(* CODESYS project tcl_SimpleUnitTestLibrary.library
   Company: Red Rock Controls Limited
   Description: Local variables in T_UnitTestBase hidden
   Version: 1.1.10.2
   Placeholder: tcl_SimpleUnitTestLibrary
   Author: Roger Christopher
   Title: tcl_SimpleUnitTestLibrary

Project tree, tasks and I/O mapping:
  libraries: Tc2_EtherCAT, * (Beckhoff Automation GmbH); Tc2_Standard, * (Beckhoff Automation GmbH); Tc2_System, * (Beckhoff Automation GmbH); Tc2_Utilities, * (Beckhoff Automation GmbH); Tc3_Module, * (Beckhoff Automation GmbH); tcl_StringUtils, * (Red Rock Controls Limited)
  GVLs/
    global variables Parameters
  Unit Test Framework/
    Assertions/
      interface I_AssertionMessageList: AddMessage, Clear
      function block T_Assertion [ST]: Assert, AssertEquals_BLOB, AssertEquals_BOOL, AssertEquals_BYTE, AssertEquals_DINT, AssertEquals_DWORD, AssertEquals_INT, AssertEquals_INTERFACE, AssertEquals_LINT, AssertEquals_LREAL, AssertEquals_PVOID, AssertEquals_REAL, AssertEquals_STRING, AssertEquals_UDINT, AssertEquals_UINT, AssertEquals_ULINT, AssertEquals_WORD, AssertNotEquals_INTERFACE, FB_init, AssertionFailed, AssertionMessage
    Message list/
      function block T_AssertionMessageList [ST]: AddMessage, Clear, FB_init
    Test Runner/
      Test Runner/
        function block T_TestRunner [ST]: AddTest, AddTestSuite, BeginTesting, ClearTests, DisableAll, EnableAll, GetEnabledTestCount, GetResultsSummary, Initialisation, ResetTests, ToggleTestEnable, Busy, ReloadTests, TestFinished
    TestSuite/
      interface I_TestSuite: AddTest, GetTest, Name, TestCount
      function block T_TestSuite [ST]: AddTest, FB_init, GetTest, Name, TestCount
    Unit Test/
      interface I_AssertionListener: OnAssertionFailed, TestName
      interface I_UnitTest: Execute, Initialise, CompletedTestsCount, FailedTestsCount, ImageRef, SuiteName, TestCompleted, TestEnabled, TestHasFailed, TestHasFinished, TestName, TestState
      function block T_UnitTestBase [ST]: Execute, FB_init, Initialise, OnAssertionFailed, setTestName, TestFinished, CompletedTestsCount, FailedTestsCount, ImageRef, SuiteName, TestCompleted, TestEnabled, TestHasFailed, TestHasFinished, TestName, TestState
    Version/
      global variables Global_Version
    data type ST_TestResult
  VISUs/
    visualisation Visualization
  GlobalImagePool
  00000000-0000-0000-0000-000000000000|Images\Failed.png
  00000000-0000-0000-0000-000000000000|Images\Passed.png
  00000000-0000-0000-0000-000000000000|Images\BlueRight.png
  text list GlobalTextList
*)

// Unit Test Framework/ST_TestResult
TYPE
    ST_TestResult :
    STRUCT
        SuiteName : T_MaxString;
        TestName  : T_MaxString;
        TestState : T_MaxString;
        ImageRef  : STRING;
    END_STRUCT
END_TYPE

// GVLs/Parameters
VAR_GLOBAL CONSTANT
    MAX_TESTS              : DINT := 200;
    MAX_ASSERTION_MESSAGES : DINT := 200;
END_VAR

// Unit Test Framework/Version/Global_Version
{attribute 'TcGenerated'}
{attribute 'no-analysis'}
{attribute 'linkalways'}
// This function has been automatically generated from the project information.
VAR_GLOBAL CONSTANT
	{attribute 'const_non_replaced'}
	stLibVersion_tcl_SimpleUnitTestLibrary : ST_LibVersion := (iMajor := 1, iMinor := 1, iBuild := 10, iRevision := 2, nFlags := 0, sVersion := '1.1.10.2');
END_VAR

// Unit Test Framework/Assertions/I_AssertionMessageList
INTERFACE I_AssertionMessageList

METHOD AddMessage : BOOL
VAR_INPUT
    Message : T_MaxString;
END_VAR
END_METHOD

METHOD Clear
VAR_INPUT
END_VAR
END_METHOD

END_INTERFACE

// Unit Test Framework/Assertions/T_Assertion
FUNCTION_BLOCK T_Assertion
VAR_INPUT
END_VAR
VAR_OUTPUT
END_VAR
VAR
    _AssertionFailed : BOOL;
    _AssertionMessage : T_MaxString;
    _ExpectedAsString : T_MaxString;
    _ActualAsString   : T_MaxString;
    _AssertionListener : I_AssertionListener;
END_VAR

METHOD Assert
VAR_INPUT
    AssertionMessage : T_MaxString;
    Expected         : T_MaxString;
    Actual           : T_MaxString;
END_VAR
_AssertionFailed := TRUE;
_AssertionMessage := F_FormatStringEx2('Assertion failed in %s - %s',_AssertionListener.TestName, AssertionMessage);
    _ExpectedAsString := F_FormatStringEx1('  Expected = %s', Expected);
    _ActualAsString   := F_FormatStringEx1('  Actual   = %s', Actual);
_AssertionListener.OnAssertionFailed(_AssertionMessage,_ExpectedAsString,_ActualAsString);
END_METHOD

METHOD AssertEquals_BLOB
VAR_INPUT
    Expected : ANY;
    Actual   : ANY;
    VariableName : T_MaxString;
END_VAR
IF Expected.diSize <> Actual.diSize THEN
    _AssertionFailed := TRUE;
    _AssertionMessage := F_FormatStringEx2('AssertEquals_BLOB failed in %s: Value "%s"', _AssertionListener.TestName, 'Blob.Size');
    _ExpectedAsString := F_FormatString1('  Expected = %d', F_DINT(Expected.diSize));
    _ActualAsString   := F_FormatString1('  Actual   = %d', F_DINT(Actual.diSize));
    _AssertionListener.OnAssertionFailed(_AssertionMessage,_ExpectedAsString,_ActualAsString);
    
ELSIF Expected.TypeClass <> Actual.TypeClass THEN
    _AssertionFailed := TRUE;
    _AssertionMessage := F_FormatStringEx2('AssertEquals_BLOB failed in %s: Value "%s"', _AssertionListener.TestName, 'Blob.TypeClass');
    _ExpectedAsString := F_FormatStringEx1('  Expected = %s', F_TypeClassToString(Expected.TypeClass));
    _ActualAsString   := F_FormatStringEx1('  Actual   = %s', F_TypeClassToString(Actual.TypeClass));
    _AssertionListener.OnAssertionFailed(_AssertionMessage,_ExpectedAsString,_ActualAsString);
    
ELSIF 
    MEMCMP(
        pBuf1 := Expected.pValue, 
        pBuf2 := Actual.pValue, 
        n     := DINT_TO_UDINT(Actual.diSize)) <> 0
THEN
    _AssertionFailed := TRUE;
    _AssertionMessage := F_FormatStringEx1('AssertEquals_BLOB failed in %s: Contents differ', _AssertionListener.TestName);
    _ExpectedAsString := '';
    _ActualAsString   := '';
    _AssertionListener.OnAssertionFailed(_AssertionMessage,_ExpectedAsString,_ActualAsString);
ELSE
    _AssertionFailed  := FALSE;
    _AssertionMessage := '';
END_IF
END_METHOD

METHOD AssertEquals_BOOL 
VAR_INPUT
    Expected : BOOL;
    Actual   : BOOL;
    VariableName : T_MaxString;
END_VAR
IF Expected <> Actual THEN
    _AssertionFailed  := TRUE;
    _AssertionMessage := F_FormatStringEx2('AssertEquals_BOOL failed in %s: Value "%s"', _AssertionListener.TestName, VariableName);
    _ExpectedAsString := F_FormatStringEx1('  Expected = %s', BOOL_TO_STRING(Expected));
    _ActualAsString   := F_FormatStringEx1('  Actual   = %s', BOOL_TO_STRING(Actual));
    _AssertionListener.OnAssertionFailed(_AssertionMessage,_ExpectedAsString,_ActualAsString);
ELSE
    _AssertionFailed   := FALSE;
    _AssertionMessage  := '';
END_IF
END_METHOD

METHOD AssertEquals_BYTE
VAR_INPUT
    Expected : BYTE;
    Actual   : BYTE;
    VariableName : T_MaxString;
END_VAR
IF Expected <> Actual THEN
    _AssertionFailed := TRUE;
    _AssertionMessage := F_FormatStringEx2('AssertEquals_BYTE failed in %s: Value "%s"', _AssertionListener.TestName, VariableName);
    _ExpectedAsString := F_FormatString1('  Expected = %d', F_BYTE(Expected));
    _ActualAsString   := F_FormatString1('  Actual   = %d', F_BYTE(Actual));
    _AssertionListener.OnAssertionFailed(_AssertionMessage,_ExpectedAsString,_ActualAsString);
ELSE
    _AssertionFailed  := FALSE;
    _AssertionMessage := '';
END_IF
END_METHOD

METHOD AssertEquals_DINT 
VAR_INPUT
    Expected : DINT;
    Actual   : DINT;
    VariableName : T_MaxString;
END_VAR
IF Expected <> Actual THEN
    _AssertionFailed  := TRUE;
    _AssertionMessage := F_FormatStringEx2('AssertEquals_DINT failed in %s: Value "%s"', _AssertionListener.TestName, VariableName);
    _ExpectedAsString := F_FormatString1('  Expected = %d', F_DINT(Expected));
    _ActualAsString   := F_FormatString1('  Actual   = %d', F_DINT(Actual));
    _AssertionListener.OnAssertionFailed(_AssertionMessage,_ExpectedAsString,_ActualAsString);
ELSE
    _AssertionFailed  := FALSE;
    _AssertionMessage := '';
END_IF
END_METHOD

METHOD AssertEquals_DWORD
VAR_INPUT
    Expected : DWORD;
    Actual   : DWORD;
    VariableName : T_MaxString;
END_VAR
IF Expected <> Actual THEN
    _AssertionFailed := TRUE;
    _AssertionMessage := F_FormatStringEx2('AssertEquals_DWORD failed in %s: Value "%s"', _AssertionListener.TestName, VariableName);
    _ExpectedAsString := F_FormatString1('  Expected = %d', F_DWORD(Expected));
    _ActualAsString   := F_FormatString1('  Actual   = %d', F_DWORD(Actual));
    _AssertionListener.OnAssertionFailed(_AssertionMessage,_ExpectedAsString,_ActualAsString);
ELSE
    _AssertionFailed  := FALSE;
    _AssertionMessage := '';
END_IF
END_METHOD

METHOD AssertEquals_INT
VAR_INPUT
    Expected : INT;
    Actual   : INT;
    VariableName : T_MaxString;
END_VAR
IF Expected <> Actual THEN
    _AssertionFailed := TRUE;
    _AssertionMessage := F_FormatStringEx2('AssertEquals_INT failed in %s: Value "%s"', _AssertionListener.TestName, VariableName);
    _ExpectedAsString := F_FormatString1('  Expected = %d', F_INT(Expected));
    _ActualAsString   := F_FormatString1('  Actual   = %d', F_INT(Actual));
    _AssertionListener.OnAssertionFailed(_AssertionMessage,_ExpectedAsString,_ActualAsString);
ELSE
    _AssertionFailed  := FALSE;
    _AssertionMessage := '';
END_IF
END_METHOD

METHOD AssertEquals_INTERFACE 
VAR_INPUT
    Expected : __SYSTEM.IQueryInterface;
    Actual   : __SYSTEM.IQueryInterface;
    VariableName : T_MaxString;
END_VAR
IF Expected <> Actual THEN
    _AssertionFailed  := TRUE;
    _AssertionMessage := F_FormatStringEx2('AssertEquals_INTERFACE failed in %s: Value "%s"', _AssertionListener.TestName, VariableName);
    _ExpectedAsString := '  Interfaces Differ';
    _ActualAsString   := '';
    _AssertionListener.OnAssertionFailed(_AssertionMessage,_ExpectedAsString,_ActualAsString);
ELSE
    _AssertionFailed  := FALSE;
    _AssertionMessage := '';
END_IF
END_METHOD

METHOD AssertEquals_LINT 
VAR_INPUT
    Expected : LINT;
    Actual   : LINT;
    VariableName : T_MaxString;
END_VAR
IF Expected <> Actual THEN
    _AssertionFailed  := TRUE;
    _AssertionMessage := F_FormatStringEx2('AssertEquals_LINT failed in %s: Value "%s"', _AssertionListener.TestName, VariableName);
    _ExpectedAsString := F_FormatString1('  Expected = %d', F_LINT(Expected));
    _ActualAsString   := F_FormatString1('  Actual   = %d', F_LINT(Actual));
    _AssertionListener.OnAssertionFailed(_AssertionMessage,_ExpectedAsString,_ActualAsString);
ELSE
    _AssertionFailed  := FALSE;
    _AssertionMessage := '';
END_IF
END_METHOD

METHOD AssertEquals_LREAL 
VAR_INPUT
    Expected : LREAL;
    Actual   : LREAL;
    Delta    : LREAL;
    VariableName : T_MaxString;
END_VAR
IF ABS(Expected - Actual) > Delta THEN
    _AssertionFailed  := TRUE;
    _AssertionMessage := F_FormatStringEx2('AssertEquals_LREAL failed in %s: Value "%s"', _AssertionListener.TestName, VariableName);
    _ExpectedAsString := F_FormatString1('  Expected = %f', F_LREAL(Expected));
    _ActualAsString   := F_FormatString1('  Actual   = %f', F_LREAL(Actual));
    _AssertionListener.OnAssertionFailed(_AssertionMessage,_ExpectedAsString,_ActualAsString);
ELSE
    _AssertionFailed  := FALSE;
    _AssertionMessage := '';
END_IF
END_METHOD

METHOD AssertEquals_PVOID 
VAR_INPUT
    Expected : PVOID;
    Actual   : PVOID;
    VariableName : T_MaxString;
END_VAR
IF Expected <> Actual THEN
    _AssertionFailed  := TRUE;
    _AssertionMessage := F_FormatStringEx2('AssertEquals_PVOID failed in %s: Value "%s"', _AssertionListener.TestName, VariableName);
    _ExpectedAsString := F_FormatString1('  Expected = %d', F_PVOID(Expected));
    _ActualAsString   := F_FormatString1('  Actual   = %d', F_PVOID(Actual));
    _AssertionListener.OnAssertionFailed(_AssertionMessage,_ExpectedAsString,_ActualAsString);
ELSE
    _AssertionFailed  := FALSE;
    _AssertionMessage := '';
END_IF
END_METHOD

METHOD AssertEquals_REAL 
VAR_INPUT
    Expected : REAL;
    Actual   : REAL;
    Delta    : REAL;
    VariableName : T_MaxString;
END_VAR
IF ABS(Expected - Actual) > Delta THEN
    _AssertionFailed  := TRUE;
    _AssertionMessage := F_FormatStringEx2('AssertEquals_REAL failed in %s: Value "%s"', _AssertionListener.TestName, VariableName);
    _ExpectedAsString := F_FormatString1('  Expected = %f', F_REAL(Expected));
    _ActualAsString   := F_FormatString1('  Actual   = %f', F_REAL(Actual));
    _AssertionListener.OnAssertionFailed(_AssertionMessage,_ExpectedAsString,_ActualAsString);
ELSE
    _AssertionFailed  := FALSE;
    _AssertionMessage := '';
END_IF
END_METHOD

METHOD AssertEquals_STRING
VAR_INPUT
    Expected : T_MaxString;
    Actual   : T_MaxString;
    VariableName : T_MaxString;
END_VAR
IF Expected <> Actual THEN
    _AssertionFailed := TRUE;
    _AssertionMessage := F_FormatStringEx2('AssertEquals_STRING failed in %s: Value "%s"', _AssertionListener.TestName, VariableName);
    _ExpectedAsString := F_FormatStringEx1('  Expected = %s', Expected);
    _ActualAsString   := F_FormatStringEx1('  Actual   = %s', Actual);
    _AssertionListener.OnAssertionFailed(_AssertionMessage,_ExpectedAsString,_ActualAsString);
ELSE
    _AssertionFailed   := FALSE;
    _AssertionMessage  := '';
    _ExpectedAsString  := '';
    _ActualAsString    := '';
END_IF
END_METHOD

METHOD AssertEquals_UDINT
VAR_INPUT
    Expected : UDINT;
    Actual   : UDINT;
    VariableName : T_MaxString;
END_VAR
IF Expected <> Actual THEN
    _AssertionFailed := TRUE;
    _AssertionMessage := F_FormatStringEx2('AssertEquals_UDINT failed in %s: Value "%s"', _AssertionListener.TestName, VariableName);
    _ExpectedAsString := F_FormatString1('  Expected = %d', F_UDINT(Expected));
    _ActualAsString   := F_FormatString1('  Actual   = %d', F_UDINT(Actual));
    _AssertionListener.OnAssertionFailed(_AssertionMessage,_ExpectedAsString,_ActualAsString);
ELSE
    _AssertionFailed  := FALSE;
    _AssertionMessage := '';
END_IF
END_METHOD

METHOD AssertEquals_UINT
VAR_INPUT
    Expected : UINT;
    Actual   : UINT;
    VariableName : T_MaxString;
END_VAR
IF Expected <> Actual THEN
    _AssertionFailed := TRUE;
    _AssertionMessage := F_FormatStringEx2('AssertEquals_UINT failed in %s: Value "%s"', _AssertionListener.TestName, VariableName);
    _ExpectedAsString := F_FormatString1('  Expected = %d', F_UINT(Expected));
    _ActualAsString   := F_FormatString1('  Actual   = %d', F_UINT(Actual));
    _AssertionListener.OnAssertionFailed(_AssertionMessage,_ExpectedAsString,_ActualAsString);
ELSE
    _AssertionFailed  := FALSE;
    _AssertionMessage := '';
END_IF
END_METHOD

METHOD AssertEquals_ULINT 
VAR_INPUT
    Expected : ULINT;
    Actual   : ULINT;
    VariableName : T_MaxString;
END_VAR
IF Expected <> Actual THEN
    _AssertionFailed  := TRUE;
    _AssertionMessage := F_FormatStringEx2('AssertEquals_ULINT failed in %s: Value "%s"', _AssertionListener.TestName, VariableName);
    _ExpectedAsString := F_FormatString1('  Expected = %d', F_ULINT(Expected));
    _ActualAsString   := F_FormatString1('  Actual   = %d', F_ULINT(Actual));
    _AssertionListener.OnAssertionFailed(_AssertionMessage,_ExpectedAsString,_ActualAsString);
ELSE
    _AssertionFailed  := FALSE;
    _AssertionMessage := '';
END_IF
END_METHOD

METHOD AssertEquals_WORD
VAR_INPUT
    Expected : WORD;
    Actual   : WORD;
    VariableName : T_MaxString;
END_VAR
IF Expected <> Actual THEN
    _AssertionFailed := TRUE;
    _AssertionMessage := F_FormatStringEx2('AssertEquals_WORD failed in %s: Value "%s"', _AssertionListener.TestName, VariableName);
    _ExpectedAsString := F_FormatString1('  Expected = %d', F_WORD(Expected));
    _ActualAsString   := F_FormatString1('  Actual   = %d', F_WORD(Actual));
    _AssertionListener.OnAssertionFailed(_AssertionMessage,_ExpectedAsString,_ActualAsString);
ELSE
    _AssertionFailed  := FALSE;
    _AssertionMessage := '';
END_IF
END_METHOD

METHOD AssertNotEquals_INTERFACE 
VAR_INPUT
    Expected : __SYSTEM.IQueryInterface;
    Actual   : __SYSTEM.IQueryInterface;
    VariableName : T_MaxString;
END_VAR
IF Expected = Actual THEN
    _AssertionFailed  := TRUE;
    _AssertionMessage := F_FormatStringEx2('AssertNotEquals_INTERFACE failed in %s: Value "%s"', _AssertionListener.TestName, VariableName);
    _ExpectedAsString := '  Interfaces are the same';
    _ActualAsString   := '';
    _AssertionListener.OnAssertionFailed(_AssertionMessage,_ExpectedAsString,_ActualAsString);
ELSE
    _AssertionFailed  := FALSE;
    _AssertionMessage := '';
END_IF
END_METHOD

METHOD FB_init : BOOL
VAR_INPUT
	bInitRetains : BOOL; // if TRUE, the retain variables are initialized (warm start / cold start)
	bInCopyCode : BOOL;  // if TRUE, the instance afterwards gets moved into the copy code (online change)
    AssertionListener : I_AssertionListener;
END_VAR
_AssertionListener := AssertionListener;
END_METHOD

PROPERTY AssertionFailed : BOOL
GET
AssertionFailed := _AssertionFailed;
END_GET
END_PROPERTY

PROPERTY AssertionMessage : T_MaxString
GET
AssertionMessage := _AssertionMessage;
END_GET
END_PROPERTY

END_FUNCTION_BLOCK

// Unit Test Framework/Unit Test/I_AssertionListener
INTERFACE I_AssertionListener

METHOD OnAssertionFailed
VAR_INPUT
    AssertionMessage : T_MaxString;
    ExpectedAsString : T_MaxString;
    ActualAsString   : T_MaxString;
END_VAR
END_METHOD

{attribute 'monitoring' := 'call'}
PROPERTY TestName : T_MaxString
GET
END_GET
END_PROPERTY

END_INTERFACE

// Unit Test Framework/Message list/T_AssertionMessageList
FUNCTION_BLOCK T_AssertionMessageList IMPLEMENTS I_AssertionMessageList
VAR
    Messages : REFERENCE TO ARRAY[0..MAX_ASSERTION_MESSAGES] OF T_MaxString;
    Count : INT;
END_VAR

METHOD AddMessage : BOOL
VAR_INPUT
    Message : T_MaxString;
END_VAR
IF Count <= MAX_ASSERTION_MESSAGES THEN
    Messages[Count] := Message;
    Count := Count + 1;
    AddMessage := TRUE;
END_IF
END_METHOD

METHOD Clear
VAR_INPUT
END_VAR
MEMSET(
    destAddr := ADR(Messages), 
    fillByte := 0, 
    n        := SIZEOF(Messages));
Count := 0;
END_METHOD

METHOD FB_init : BOOL
VAR_INPUT
    bInitRetains : BOOL; // if TRUE, the retain variables are initialized (warm start / cold start)
    bInCopyCode  : BOOL; // if TRUE, the instance afterwards gets moved into the copy code (online change)
    Messages     : REFERENCE TO ARRAY[0..MAX_ASSERTION_MESSAGES] OF T_MaxString;
END_VAR
THIS^.Messages REF= Messages;
END_METHOD

END_FUNCTION_BLOCK

// Unit Test Framework/Test Runner/Test Runner/T_TestRunner
FUNCTION_BLOCK T_TestRunner
VAR
    _ReloadTests         : BOOL := TRUE; // Also exposed as a property so it can be read and reset by client
    RunTestsSequentially : BOOL := TRUE;
    Run                  : BOOL;
    Reset                : BOOL;
    EnableAllTests       : BOOL;
    DisableAllTests      : BOOL;
    RowIsSelected        : BOOL;
    SelectedRow          : INT := -1;
    Abort                : BOOL;

    State : (
        Init,
        StartTests,
        RunTests_Concurrently,
        RunTests_Sequentially,
        CheckResults
    );

    i                        : DINT;
    CompletedTestsCount      : DINT;
    FailedTestsCount         : DINT;
    CurrentTestIndex         : DINT;
    TestsCompletedPercentage : LREAL;
    TestCount                : DINT;
    EnabledTestCount         : DINT;
    ResultsSummary           : T_MaxString;

    Results  : ARRAY[0..MAX_TESTS] OF ST_TestResult;
    Tests    : ARRAY[0..MAX_TESTS] OF I_UnitTest;
    Messages : ARRAY[0..MAX_ASSERTION_MESSAGES] OF T_MaxString; // must be located here so vis can access them

    AssertionMessages : T_AssertionMessageList(Messages := Messages);

END_VAR

IF RowIsSelected THEN
    ToggleTestEnable(Index := SelectedRow);
    RowIsSelected := FALSE;
	SelectedRow := -1;
END_IF

IF EnableAllTests THEN
    EnableAllTests := FALSE;
    EnableAll();
END_IF

IF DisableAllTests THEN
    DisableAllTests := FALSE;
    DisableAll();
END_IF

IF Abort THEN
	Abort := FALSE;
	State := 0;
	Initialisation();
END_IF

CASE State OF
    Init:
        IF Reset THEN
            Reset := FALSE;
            Initialisation();
        END_IF

        IF Run THEN
            Run              := FALSE;
            EnabledTestCount := GetEnabledTestCount();

            IF EnabledTestCount = 0 THEN
                State := CheckResults;
            ELSE
                State := StartTests;
            END_IF
        END_IF

    StartTests:
        IF RunTestsSequentially THEN
            State := RunTests_Sequentially;
        ELSE
            State := RunTests_Concurrently;
        END_IF

    RunTests_Concurrently:
        FOR i := 0 TO TestCount - 1 DO
            Tests[i].Execute();
			Results[i].TestState := Tests[i].TestState;
			Results[i].ImageRef  := Tests[i].ImageRef;
        END_FOR

        IF EnabledTestCount > 0 THEN
            TestsCompletedPercentage := CompletedTestsCount * 100 / EnabledTestCount;
        END_IF

        ResultsSummary := GetResultsSummary();

        IF CompletedTestsCount >= EnabledTestCount THEN
            State := CheckResults;
        END_IF

    RunTests_Sequentially:
        IF Tests[CurrentTestIndex] <> 0 THEN
            Tests[CurrentTestIndex].Execute();
			Results[CurrentTestIndex].TestState := Tests[CurrentTestIndex].TestState;
			Results[CurrentTestIndex].ImageRef  := Tests[CurrentTestIndex].ImageRef;

            IF NOT Tests[CurrentTestIndex].TestEnabled OR Tests[CurrentTestIndex].TestHasFinished THEN
                CurrentTestIndex := CurrentTestIndex + 1;
            END_IF
        END_IF

        IF EnabledTestCount > 0 THEN
            TestsCompletedPercentage := CompletedTestsCount * 100 / EnabledTestCount;
        END_IF

        ResultsSummary := GetResultsSummary();

        IF CurrentTestIndex >= TestCount THEN
            State := CheckResults;
        END_IF

    CheckResults:
        ResultsSummary := GetResultsSummary();
        State          := Init;

END_CASE

METHOD AddTest : BOOL
VAR_INPUT
    UnitTest : I_UnitTest;
END_VAR
IF TestCount < MAX_TESTS THEN
    UnitTest.TestEnabled := TRUE;
    Tests[TestCount]    := UnitTest;
	    Results[TestCount].SuiteName := UnitTest.SuiteName;
	    Results[TestCount].TestName  := UnitTest.TestName;
	    Results[TestCount].TestState := UnitTest.TestState;
	    Results[TestCount].ImageRef  := UnitTest.ImageRef;
	
    TestCount           := TestCount + 1;
    AddTest              := TRUE;
ELSE
    AssertionMessages.AddMessage('Maximum unit tests exceeded!');
END_IF
END_METHOD

METHOD AddTestSuite : BOOL
VAR_INPUT
    TestSuite : I_TestSuite;
END_VAR
VAR
    i : INT;
    UnitTestToAdd : I_UnitTest;
END_VAR
IF TestSuite.TestCount > 0 THEN
    FOR i := 0 TO TestSuite.TestCount - 1 DO
        UnitTestToAdd := TestSuite.GetTest(i);
        AddTest(UnitTestToAdd);
    END_FOR
END_IF
END_METHOD

METHOD PUBLIC BeginTesting : BOOL
IF state <> init THEN
  RETURN;
END_IF

Run := TRUE;
BeginTesting := TRUE;
END_METHOD

METHOD ClearTests
VAR_INPUT
END_VAR
FOR i := 0 TO MAX_TESTS DO
    Tests[i] := 0;
END_FOR
MEMSET(
	destAddr:= ADR(Results), 
	fillByte:= 0, 
	n:= SIZEOF(Results));
TestCount := 0;
END_METHOD

METHOD DisableAll
VAR_INPUT
END_VAR
IF State = Init THEN
    FOR i := 0 TO MAX_TESTS - 1 DO
        IF Tests[i] <> 0 THEN
            Tests[i].TestEnabled := FALSE;
			Results[i].TestState := 'Disabled';
        END_IF
    END_FOR
END_IF
END_METHOD

METHOD EnableAll
VAR_INPUT
END_VAR
IF State = Init THEN
    FOR i := 0 TO MAX_TESTS - 1 DO
        IF Tests[i] <> 0 THEN
            Tests[i].TestEnabled := TRUE;
			Results[i].TestState := 'Enabled';
        END_IF
    END_FOR
END_IF
END_METHOD

METHOD GetEnabledTestCount : DINT
VAR
    i : DINT;
END_VAR
FOR i := 0 TO MAX_TESTS - 1 DO
    IF Tests[i] <> 0 THEN
        IF Tests[i].TestEnabled THEN
            GetEnabledTestCount := GetEnabledTestCount + 1;
        END_IF
    END_IF
END_FOR
END_METHOD

METHOD GetResultsSummary : T_MaxString
VAR_INPUT
END_VAR
GetResultsSummary := F_FormatString3('%d Tests of %d completed, %d Tests Failed',
                            F_DINT(CompletedTestsCount),
                            F_DINT(EnabledTestCount),
                            F_DINT(FailedTestsCount));
END_METHOD

METHOD Initialisation
VAR_INPUT
END_VAR
VAR
    i : DINT;
END_VAR
FOR i := 0 TO MAX_TESTS DO
    IF Tests[i] <> 0 THEN
        Tests[i].Initialise(AssertionMessages,
                            CompletedTestsCount := CompletedTestsCount,
                            FailedTestsCount    := FailedTestsCount);
							
	    Results[i].SuiteName := Tests[i].SuiteName;
	    Results[i].TestName  := Tests[i].TestName;
	    Results[i].TestState := Tests[i].TestState;
	    Results[i].ImageRef  := Tests[i].ImageRef;
    END_IF
END_FOR

ResultsSummary           := '';
FailedTestsCount         := 0;
CompletedTestsCount      := 0;
TestsCompletedPercentage := 0;
CurrentTestIndex         := 0;
AssertionMessages.Clear();
END_METHOD

METHOD PUBLIC ResetTests : BOOL
VAR_INPUT
END_VAR
IF state <> Init THEN
  RETURN;
END_IF

Reset := TRUE;
ResetTests := TRUE;
END_METHOD

METHOD ToggleTestEnable
VAR_INPUT
    Index : INT;
END_VAR
IF State = Init THEN
	IF Tests[Index].TestEnabled THEN
		Tests[Index].TestEnabled := FALSE;
		Results[Index].TestState := 'Disabled';
	ELSE
		Tests[Index].TestEnabled := TRUE;
		Results[Index].TestState := 'Enabled';
	END_IF
END_IF
END_METHOD

PROPERTY PUBLIC Busy : BOOL
GET
Busy := (State <> Init);
END_GET
END_PROPERTY

//{attribute 'monitoring' := 'call'}
PROPERTY ReloadTests : BOOL
GET
ReloadTests := _ReloadTests;
END_GET
SET
_ReloadTests := ReloadTests;
END_SET
END_PROPERTY

PROPERTY PUBLIC TestFinished : BOOL
GET
TestFinished := (CurrentTestIndex >= TestCount);
END_GET
END_PROPERTY

END_FUNCTION_BLOCK

// Unit Test Framework/Unit Test/I_UnitTest
INTERFACE I_UnitTest EXTENDS __SYSTEM.IQueryInterface

METHOD Execute
END_METHOD

METHOD Initialise
VAR_INPUT
    MessageList         : I_AssertionMessageList;
    CompletedTestsCount : REFERENCE TO DINT;
    FailedTestsCount    : REFERENCE TO DINT;
END_VAR
END_METHOD

PROPERTY CompletedTestsCount : REFERENCE TO DINT
GET
END_GET
SET
END_SET
END_PROPERTY

PROPERTY FailedTestsCount : REFERENCE TO DINT
GET
END_GET
SET
END_SET
END_PROPERTY

{attribute 'monitoring' := 'call'}
PROPERTY ImageRef : T_MaxString
GET
END_GET
SET
END_SET
END_PROPERTY

{attribute 'monitoring' := 'call'}
PROPERTY SuiteName : T_MaxString
GET
END_GET
END_PROPERTY

PROPERTY TestCompleted : BOOL
GET
END_GET
SET
END_SET
END_PROPERTY

{attribute 'monitoring' := 'call'}
PROPERTY TestEnabled : BOOL
GET
END_GET
SET
END_SET
END_PROPERTY

PROPERTY TestHasFailed : BOOL
GET
END_GET
SET
END_SET
END_PROPERTY

PROPERTY TestHasFinished : BOOL
GET
END_GET
SET
END_SET
END_PROPERTY

{attribute 'monitoring' := 'call'}
PROPERTY TestName : T_MaxString
GET
END_GET
END_PROPERTY

{attribute 'monitoring' := 'call'}
PROPERTY TestState : T_MaxString
GET
END_GET
SET
END_SET
END_PROPERTY

END_INTERFACE

// Unit Test Framework/TestSuite/I_TestSuite
INTERFACE I_TestSuite

METHOD AddTest : BOOL
VAR_INPUT
    UnitTest : I_UnitTest;
END_VAR
END_METHOD

METHOD GetTest : I_UnitTest
VAR_INPUT
    Index : INT;
END_VAR
END_METHOD

PROPERTY Name : T_MaxString
GET
END_GET
END_PROPERTY

PROPERTY TestCount : INT
GET
END_GET
END_PROPERTY

END_INTERFACE

// Unit Test Framework/TestSuite/T_TestSuite
{attribute 'reflection'}
FUNCTION_BLOCK T_TestSuite IMPLEMENTS I_TestSuite
VAR_INPUT
END_VAR
VAR_OUTPUT
END_VAR
VAR
    {attribute 'instance-path'} 
    {attribute 'no_init'}
    _TestSuiteName       : T_MaxString; // Automatically initialised with the full name of the instance
    _TestCount : INT;
    Tests : ARRAY[0..MAX_TESTS_PER_TEST_SUITE] OF I_UnitTest;
END_VAR
VAR CONSTANT
    MAX_TESTS_PER_TEST_SUITE              : DINT := 100;
END_VAR

METHOD AddTest : BOOL
VAR_INPUT
    UnitTest : I_UnitTest;
END_VAR
IF _TestCount < MAX_TESTS_PER_TEST_SUITE THEN
    Tests[_TestCount] := UnitTest;
    _TestCount := _TestCount + 1;
    AddTest := TRUE;
END_IF
END_METHOD

METHOD FB_init : BOOL
VAR_INPUT
	bInitRetains : BOOL; // if TRUE, the retain variables are initialized (warm start / cold start)
	bInCopyCode : BOOL;  // if TRUE, the instance afterwards gets moved into the copy code (online change)
END_VAR
VAR
    StringSplitter : T_StringSplitter;
END_VAR
StringSplitter.Init(
    Str := _TestSuiteName,
    Delim1 := '.',
    Delim2 := '');
    
WHILE StringSplitter.HasMore() DO
    _TestSuiteName := StringSplitter.GetNext(); // to get last sub-section
END_WHILE
END_METHOD

METHOD GetTest : I_UnitTest
VAR_INPUT
    Index : INT;
END_VAR
IF Index >= 0 AND Index < _TestCount THEN
    GetTest := Tests[Index];
END_IF
END_METHOD

PROPERTY Name : T_MaxString
GET
Name := _TestSuiteName;
END_GET
END_PROPERTY

PROPERTY TestCount : INT
GET
TestCount := _TestCount;
END_GET
END_PROPERTY

END_FUNCTION_BLOCK

// Unit Test Framework/Unit Test/T_UnitTestBase
{attribute 'reflection'}
{attribute 'hide_all_locals'}
FUNCTION_BLOCK ABSTRACT T_UnitTestBase IMPLEMENTS I_UnitTest, I_AssertionListener
VAR
    {attribute 'instance-path'}
    {attribute 'no_init'}
    _InstanceName  : T_MaxString; // Automatically initialised with the full name of the instance
    _TestSuiteName : T_MaxString;
    _TestName      : T_MaxString;
    _TestFailed    : BOOL;
    _TestFinished  : BOOL;
    _TestState     : T_MaxString;
    _ImageRef      : STRING;
    _TestEnabled   : BOOL := TRUE;
    _TestCompleted : BOOL;

    _MessageList : I_AssertionMessageList;

    Assertion : T_Assertion(AssertionListener := THIS^); // Callback to allow the Assertion to update the message list on assertion failed

    _CompletedTestsCount : REFERENCE TO DINT;
    _FailedTestsCount    : REFERENCE TO DINT;
	
	State : INT; // for general use during test...
END_VAR

METHOD Execute
IF NOT TestEnabled THEN
    TestState := 'Disabled';
    ImageRef  := '';
ELSE
    IF NOT TestHasFinished THEN
        THIS^();
        IF TestHasFinished THEN
            TestCompleted := TRUE;
            CompletedTestsCount := CompletedTestsCount + 1;
            IF TestHasFailed THEN
                TestState := 'Failed';
                ImageRef  := '3';
                FailedTestsCount := FailedTestsCount + 1;
            ELSE
                TestState := 'Passed';
                ImageRef  := '2';
            END_IF
        ELSE
            TestState := 'Running';
            ImageRef  := '1';
        END_IF
    END_IF
END_IF
END_METHOD

METHOD FB_init : BOOL
VAR_INPUT
	bInitRetains : BOOL; // if TRUE, the retain variables are initialized (warm start / cold start)
	bInCopyCode : BOOL;  // if TRUE, the instance afterwards gets moved into the copy code (online change)
    TestSuite : I_TestSuite;
END_VAR
IF TestSuite <> 0 THEN
    IF NOT bInCopyCode THEN // not an online change...
        THIS^._TestSuiteName := TestSuite.Name;
        THIS^.setTestName();
        TestSuite.AddTest(THIS^);
    END_IF
END_IF
END_METHOD

METHOD Initialise
VAR_INPUT
    MessageList : I_AssertionMessageList;
    CompletedTestsCount      : REFERENCE TO DINT;
    FailedTestsCount         : REFERENCE TO DINT;
END_VAR
_TestCompleted       := FALSE;
_TestFailed          := FALSE;
_TestFinished        := FALSE;
_TestState           := '';
_ImageRef            := '';
_ImageRef            := '0';
_MessageList         := MessageList;
_CompletedTestsCount REF= CompletedTestsCount;
_FailedTestsCount    REF= FailedTestsCount;

IF _TestEnabled THEN
    _TestState := 'Enabled';
ELSE
    _TestState := 'Disabled';
END_IF

State := 0;
END_METHOD

METHOD OnAssertionFailed
VAR_INPUT
    AssertionMessage : T_MaxString;
    ExpectedAsString : T_MaxString;
    ActualAsString   : T_MaxString;
END_VAR
_TestFailed := TRUE;
_MessageList.AddMessage(AssertionMessage);

IF ExpectedAsString <> '' THEN
    _MessageList.AddMessage(ExpectedAsString);
END_IF

IF ActualAsString <> '' THEN
    _MessageList.AddMessage(ActualAsString);
END_IF
END_METHOD

METHOD setTestName
VAR
    StringSplitter : T_StringSplitter;
END_VAR
StringSplitter.Init(
    Str := _InstanceName,
    Delim1 := '.',
    Delim2 := '');
    
WHILE StringSplitter.HasMore() DO
    _TestName := StringSplitter.GetNext(); // to get last sub-section
END_WHILE
END_METHOD

METHOD TestFinished
VAR_INPUT
END_VAR
_TestFinished := TRUE;
END_METHOD

PROPERTY CompletedTestsCount : REFERENCE TO DINT
GET
CompletedTestsCount REF= _CompletedTestsCount;
END_GET
SET
_CompletedTestsCount REF= CompletedTestsCount;
END_SET
END_PROPERTY

PROPERTY FailedTestsCount : REFERENCE TO DINT
GET
FailedTestsCount REF= _FailedTestsCount;
END_GET
SET
_FailedTestsCount REF= FailedTestsCount;
END_SET
END_PROPERTY

{attribute 'monitoring' := 'call'}
PROPERTY ImageRef : T_MaxString
GET
ImageRef := _ImageRef;
END_GET
SET
_ImageRef := ImageRef;
END_SET
END_PROPERTY

{attribute 'monitoring' := 'call'}
PROPERTY SuiteName : T_MaxString
GET
SuiteName := _TestSuiteName;
END_GET
END_PROPERTY

PROPERTY TestCompleted : BOOL
GET
TestCompleted := _TestCompleted;
END_GET
SET
_TestCompleted := TestCompleted;
END_SET
END_PROPERTY

{attribute 'monitoring' := 'call'}
PROPERTY TestEnabled : BOOL
GET
TestEnabled := _TestEnabled;
END_GET
SET
_TestEnabled := TestEnabled;
IF TestEnabled THEN
    _TestState := 'Enabled';
ELSE
    _TestState := 'Disabled';
END_IF
END_SET
END_PROPERTY

PROPERTY TestHasFailed : BOOL
GET
TestHasFailed := _TestFailed;
END_GET
SET
_TestFailed := TestHasFailed;
END_SET
END_PROPERTY

PROPERTY TestHasFinished : BOOL
GET
TestHasFinished := _TestFinished;
END_GET
SET
_TestFinished := TestHasFinished;
END_SET
END_PROPERTY

{attribute 'monitoring' := 'call'}
PROPERTY TestName : T_MaxString
GET
TestName := _TestName;
END_GET
END_PROPERTY

{attribute 'monitoring' := 'call'}
PROPERTY TestState : T_MaxString
GET
TestState := _TestState;
END_GET
SET
_TestState := TestState;
END_SET
END_PROPERTY

END_FUNCTION_BLOCK

// VISUs/Visualization
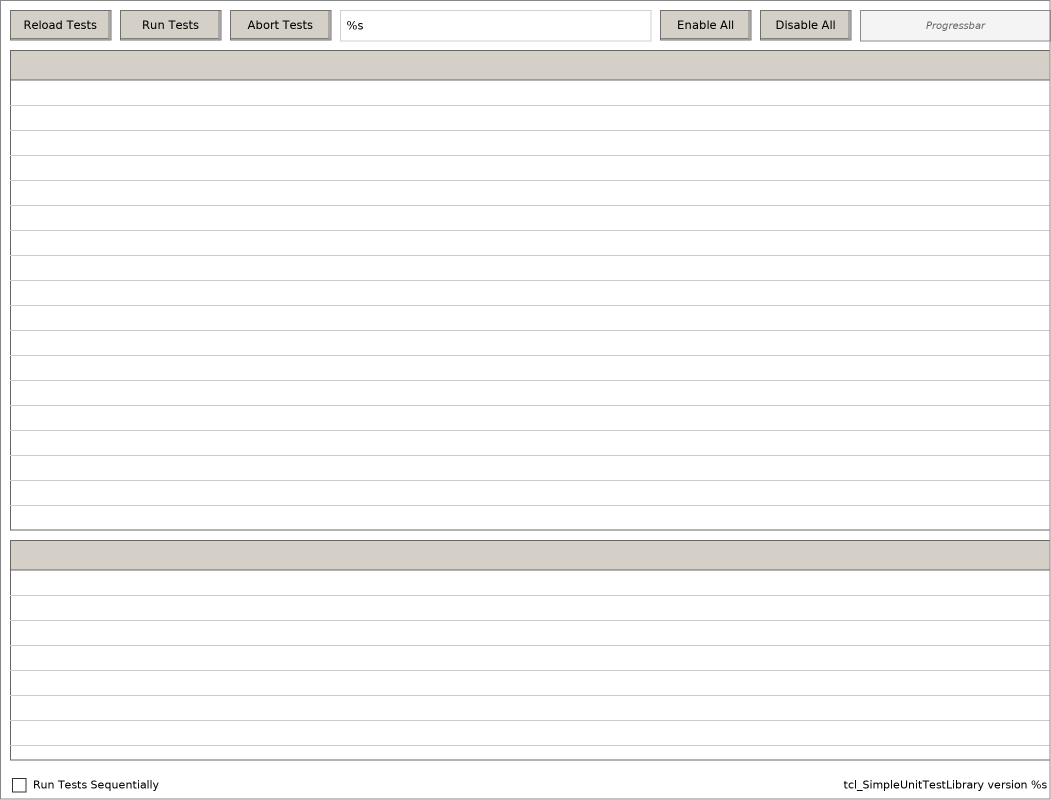
VISUALIZATION Visualization  // 1051x800
VAR_IN_OUT
    TestRunner : T_TestRunner;
END_VAR
    Button (120,10 101x30), "Run Tests"
        OnMouseDown: execute { TestRunner.Reset := TRUE; }
        OnMouseUp: execute { TestRunner.Run := TRUE; }
    Textfield (340,10 311x31), "%s", text variable: TestRunner.ResultsSummary
    Progressbar (860,10 191x31), variable: TestRunner.TestsCompletedPercentage
    Rectangle (400,770 650x30), "tcl_SimpleUnitTestLibrary version %s", text variable: Global_Version.stLibVersion_tcl_SimpleUnitTestLibrary.sVersion
    Table (10,540 1040x220), data array: TestRunner.Messages
        p1892666644: TestRunner.AssertionMessages._Count
        p1128707560: TestRunner.AssertionMessages.Count - 1
        p3854506369: TestRunner.Messages[INDEX]
        p2232123230: Assertion Messages
    Checkbox (10,770 261x30), "Run Tests Sequentially", variable: TestRunner.RunTestsSequentially
    Button (660,10 91x30), "Enable All"
        tap TestRunner.EnableAllTests
    Button (760,10 91x30), "Disable All"
        tap TestRunner.DisableAllTests
    Button (10,10 101x30), "Reload Tests"
        tap TestRunner._ReloadTests
    Table (10,50 1040x480), data array: TestRunner.Results
        p3854506369: TestRunner.Results[INDEX].ImageRef
        p1892666644: TestRunner.Results[INDEX].SuiteName
        p338671338: TestRunner.Results[INDEX].TestName
        p2170511999: TestRunner.Results[INDEX].TestState
        p1128707560: TestRunner.TestCount - 1
        p1137915858: TestRunner.SelectedRow
        p1822360349: TestRunner.RowIsSelected
    Button (230,10 101x30), "Abort Tests"
        tap TestRunner.Abort
END_VISUALIZATION
